{attribute 'qualified_only'}
{attribute 'strict'}
TYPE E_SCANNER_State :
(
	IDLE,
	CONNECT,
	SEND,
	RECEIVE,
	DISCONNECT,
	CHECKOS,
	BROWSE,
	IMAGE,
	DECODE,
	HEARTBEAT,
	DONE
);
END_TYPE

(* stored: Version 1.1.0.1
   DUT E_SCANNER_State: Id {0a70c102-1835-4b5c-a362-4f1240b3d440} *)
